{attribute 'GeneratedUsingTerminal: EL3611-1030-0016'}
{attribute addProperty BoxType "EL3611-1030-0016"}
{attribute addProperty Description "EL3611-1030 1Ch. Ana. Input 0-20 mA, Diff. 24bit"}
{attribute addProperty Physics "KK"}
{attribute addProperty Id "AI_InputsAT %I*AI_Inputs_4521310411WcStateAT %I*WcState_9091E0EB2InfoDataAT %I*InfoData_32EB74EA10"}
{attribute addProperty CRC "1887163282"}
{attribute addProperty Size "23"}
TYPE EL3611_707BD392 EXTENDS EtcSlaveTerminalBase_947E5A46 :
STRUCT
	{attribute addProperty Name "AI_Inputs"}
	AI_Inputs : AI_Inputs_45213104;
	{attribute addProperty Name "WcState"}
	WcState : WcState_9091E0EB;
	{attribute addProperty Name "InfoData"}
	InfoData : InfoData_32EB74EA;
END_STRUCT
END_TYPE

(* stored: Version 1.2.0.0, ProductVersion 3.1.4024.11
   DUT EL3611_707BD392: Id {a7439d39-3a98-4719-9184-56b26d8ea527} *)
